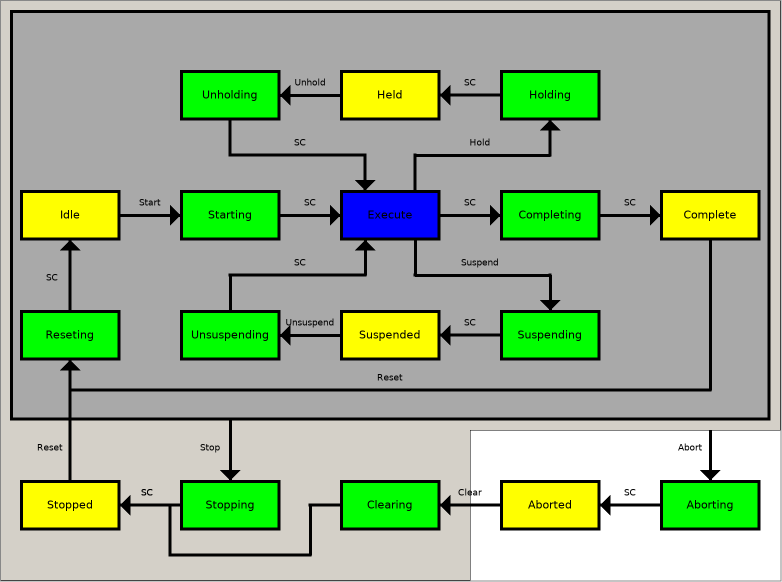
VISUALIZATION VIS_TemplatePMLStateModel  // 782x582
VAR_INPUT
	ePMLUnitMode		: DINT;
	ePMLState			: DINT;
END_VAR
    Polygon (0,0) (780,0) (780,430) (470,430) (470,580) (0,580)
    Rectangle (10,10 760x410)
    Polyline (415,190) (415,155) (550,155) (550,95) (440,95), invisible if: stPMLUnitModeConfiguration[ePMLUnitMode].aStateDisabled[11]
    Polyline (365,190) (365,155) (230,155) (230,95) (340,95), invisible if: stPMLUnitModeConfiguration[ePMLUnitMode].aStateDisabled[11]
    Polyline (415,240) (415,275) (550,275) (550,335) (440,335), invisible if: stPMLUnitModeConfiguration[ePMLUnitMode].aStateDisabled[5]
    Polyline (365,240) (365,275) (230,275) (230,335) (340,335), invisible if: stPMLUnitModeConfiguration[ePMLUnitMode].aStateDisabled[5]
    Polyline (710,430) (710,505) (310,505) (310,555) (170,555) (170,505) (70,505) (70,215) (340,215)
    RoundedRectangle (20,190 100x50), "Idle", colour toggle: (ePMLState = 4), invisible if: stPMLUnitModeConfiguration[ePMLUnitMode].aStateDisabled[4]
    RoundedRectangle (180,190 100x50), "Starting", colour toggle: (ePMLState = 3), invisible if: stPMLUnitModeConfiguration[ePMLUnitMode].aStateDisabled[3]
    RoundedRectangle (340,190 100x50), "Execute", colour toggle: (ePMLState = 6)
    RoundedRectangle (180,70 100x50), "Unholding", colour toggle: (ePMLState = 12), invisible if: stPMLUnitModeConfiguration[ePMLUnitMode].aStateDisabled[12]
    RoundedRectangle (340,70 100x50), "Held", colour toggle: (ePMLState = 11), invisible if: stPMLUnitModeConfiguration[ePMLUnitMode].aStateDisabled[11]
    RoundedRectangle (500,70 100x50), "Holding", colour toggle: (ePMLState = 10), invisible if: stPMLUnitModeConfiguration[ePMLUnitMode].aStateDisabled[10]
    RoundedRectangle (180,310 100x50), "Unsuspending", colour toggle: (ePMLState = 14), invisible if: stPMLUnitModeConfiguration[ePMLUnitMode].aStateDisabled[14]
    RoundedRectangle (340,310 100x50), "Suspended", colour toggle: (ePMLState = 5), invisible if: stPMLUnitModeConfiguration[ePMLUnitMode].aStateDisabled[5]
    RoundedRectangle (500,310 100x50), "Suspending", colour toggle: (ePMLState = 13), invisible if: stPMLUnitModeConfiguration[ePMLUnitMode].aStateDisabled[13]
    RoundedRectangle (20,310 100x50), "Reseting", colour toggle: (ePMLState = 15), invisible if: stPMLUnitModeConfiguration[ePMLUnitMode].aStateDisabled[15]
    RoundedRectangle (20,480 100x50), "Stopped", colour toggle: (ePMLState = 2)
    RoundedRectangle (340,480 100x50), "Clearing", colour toggle: (ePMLState = 1), invisible if: stPMLUnitModeConfiguration[ePMLUnitMode].aStateDisabled[1]
    RoundedRectangle (500,480 100x50), "Aborted", colour toggle: (ePMLState = 9)
    RoundedRectangle (660,480 100x50), "Aborting", colour toggle: (ePMLState = 8), invisible if: stPMLUnitModeConfiguration[ePMLUnitMode].aStateDisabled[8]
    Polygon (550,120) (540,130) (560,130), invisible if: stPMLUnitModeConfiguration[ePMLUnitMode].aStateDisabled[10]
    Polygon (365,240) (355,250) (375,250), invisible if: stPMLUnitModeConfiguration[ePMLUnitMode].aStateDisabled[5]
    Polygon (70,240) (60,250) (80,250), invisible if: stPMLUnitModeConfiguration[ePMLUnitMode].aStateDisabled[4]
    Polygon (70,360) (60,370) (80,370), invisible if: stPMLUnitModeConfiguration[ePMLUnitMode].aStateDisabled[15]
    Polygon (440,95) (450,105) (450,85), invisible if: stPMLUnitModeConfiguration[ePMLUnitMode].aStateDisabled[11]
    Polygon (280,95) (290,105) (290,85), invisible if: stPMLUnitModeConfiguration[ePMLUnitMode].aStateDisabled[12]
    Polygon (440,335) (450,345) (450,325), invisible if: stPMLUnitModeConfiguration[ePMLUnitMode].aStateDisabled[5]
    Polygon (280,335) (290,345) (290,325), invisible if: stPMLUnitModeConfiguration[ePMLUnitMode].aStateDisabled[14]
    Polygon (600,505) (610,515) (610,495)
    Polygon (440,505) (450,515) (450,495), invisible if: stPMLUnitModeConfiguration[ePMLUnitMode].aStateDisabled[1]
    Polygon (120,505) (130,515) (130,495)
    Polygon (180,215) (170,225) (170,205), invisible if: stPMLUnitModeConfiguration[ePMLUnitMode].aStateDisabled[3]
    Polygon (340,215) (330,225) (330,205)
    Polygon (500,215) (490,225) (490,205), invisible if: stPMLUnitModeConfiguration[ePMLUnitMode].aStateDisabled[16]
    Polygon (660,215) (650,225) (650,205), invisible if: stPMLUnitModeConfiguration[ePMLUnitMode].aStateDisabled[17]
    Polygon (375,180) (365,190) (355,180), invisible if: stPMLUnitModeConfiguration[ePMLUnitMode].aStateDisabled[11]
    Polygon (560,300) (550,310) (540,300), invisible if: stPMLUnitModeConfiguration[ePMLUnitMode].aStateDisabled[13]
    Polygon (720,470) (710,480) (700,470), invisible if: stPMLUnitModeConfiguration[ePMLUnitMode].aStateDisabled[8]
    Polygon (240,470) (230,480) (220,470), invisible if: stPMLUnitModeConfiguration[ePMLUnitMode].aStateDisabled[7]
    Polyline (230,420) (230,505) (150,505)
    RoundedRectangle (180,480 100x50), "Stopping", colour toggle: (ePMLState = 7), invisible if: stPMLUnitModeConfiguration[ePMLUnitMode].aStateDisabled[7]
    Label (440,135 80x15), "Hold", invisible if: stPMLUnitModeConfiguration[ePMLUnitMode].aStateDisabled[11]
    Label (260,135 80x15), "SC", invisible if: stPMLUnitModeConfiguration[ePMLUnitMode].aStateDisabled[12]
    Label (430,75 80x15), "SC", invisible if: stPMLUnitModeConfiguration[ePMLUnitMode].aStateDisabled[10]
    Label (270,75 80x15), "Unhold", invisible if: stPMLUnitModeConfiguration[ePMLUnitMode].aStateDisabled[11]
    Label (270,315 80x15), "Unsuspend", invisible if: stPMLUnitModeConfiguration[ePMLUnitMode].aStateDisabled[5]
    Label (430,315 80x15), "SC", invisible if: stPMLUnitModeConfiguration[ePMLUnitMode].aStateDisabled[13]
    Label (440,255 80x15), "Suspend", invisible if: stPMLUnitModeConfiguration[ePMLUnitMode].aStateDisabled[5]
    Label (260,255 80x15), "SC", invisible if: stPMLUnitModeConfiguration[ePMLUnitMode].aStateDisabled[14]
    Label (270,195 80x15), "SC", invisible if: stPMLUnitModeConfiguration[ePMLUnitMode].aStateDisabled[3]
    Label (590,195 80x15), "SC", invisible if: stPMLUnitModeConfiguration[ePMLUnitMode].aStateDisabled[16]
    Label (430,195 80x15), "SC", invisible if: stPMLUnitModeConfiguration[ePMLUnitMode].aStateDisabled[17]
    Label (430,485 80x15), "Clear"
    Label (590,485 80x15), "SC", invisible if: stPMLUnitModeConfiguration[ePMLUnitMode].aStateDisabled[8]
    Label (107,485 80x15), "SC", invisible if: stPMLUnitModeConfiguration[ePMLUnitMode].aStateDisabled[1]
    Label (350,370 80x15), "Reset", invisible if: stPMLUnitModeConfiguration[ePMLUnitMode].aStateDisabled[17]
    Label (10,440 80x15), "Reset", invisible if: stPMLUnitModeConfiguration[ePMLUnitMode].aStateDisabled[4]
    Label (170,440 80x15), "Stop"
    Label (650,440 80x15), "Abort"
    Label (12,270 80x15), "SC", invisible if: stPMLUnitModeConfiguration[ePMLUnitMode].aStateDisabled[15]
    Label (110,195 80x15), "Start"
    Label (107,485 80x15), "SC", invisible if: stPMLUnitModeConfiguration[ePMLUnitMode].aStateDisabled[7]
    Polyline (440,215) (710,215) (710,390) (70,390), invisible if: stPMLUnitModeConfiguration[ePMLUnitMode].aStateDisabled[17]
    RoundedRectangle (660,190 100x50), "Complete", colour toggle: (ePMLState = 17), invisible if: stPMLUnitModeConfiguration[ePMLUnitMode].aStateDisabled[17]
    RoundedRectangle (500,190 100x50), "Completing", colour toggle: (ePMLState = 16), invisible if: stPMLUnitModeConfiguration[ePMLUnitMode].aStateDisabled[16]
END_VISUALIZATION

(* stored: Version 1.1.0.1
   Visu VIS_TemplatePMLStateModel: Id {4cf49023-0575-4d13-ac94-deebcaff7985} *)
